// TIA Portal V19 export
FUNCTION_BLOCK "TYPIC_C103_BF_LSK"   // FB21, FBD
TITLE = TYPIC_C103_BF_LSK: Laagspanning koker
{ S7_Optimized_Access := 'TRUE' }
AUTHOR : OCOTECH
FAMILY : Typical
NAME : C103.801
// Logisch Object Besturing: C103.801
// 
// Het doel van de BF LSK (laagspanning koker) is om de algemene opvolging te voorzien van de laagspanningsinstallatie per verkeerskoker.
// stored: MemoryReserve 10, SetENOAutomatically false
   VAR_INPUT
      STU_ALG_LCK_SIG { ExternalAccessible := 'False'; ExternalVisible := 'False'; ExternalWritable := 'False'} : USInt;   // Onderdruk alarmen
   END_VAR
   VAR_IN_OUT
      VAR_REL : Array[0..1] of Bool;   // Array met de standmeldingen van alle vermogenschakelaars
   END_VAR
   VAR
      SIG { ExternalWritable := 'False'} : Struct   // Signaleringen
         AA01 : Bool;   // Laagspanningsinstallatie niet observeerbaar
         AA02 : Bool;   // Laagspanningsinstallatie storing algemeen
         A001 : Bool;   // Laagspanningsinstallatie standmelding beveiliging uit
         AB01 : Bool;   // Laagspanningsinstallatie niet beschikbaar
         AB02 : Bool;   // Laagspanningsinstallatie beperkt beschikbaar
      END_STRUCT;
      VAR { ExternalWritable := 'False'} : Struct   // Variabelen
         BSC : USInt;   // Geeft de beschikbaarheid aan van het deelsysteem
         LSK_STS : USInt;   // De status van het deelsysteem
         VGV_SIG_VOP : Bool;   // TRUE = Signaleringen vrijgegeven voor verkeersoperator FALSE = Onderdrukt
      END_STRUCT;
   END_VAR
BEGIN

REGION Network 1: START
END_REGION

REGION Network 2: +++ Bepalen beschikbaarheidsstatus +++
   // Beschikbaarheidsstatus (beschikbaar / beperkt beschikbaar / niet beschikbaar) bepalen.
END_REGION

REGION Network 3 (SCL): Beschikbaarheidsstatus bepalen
   IF 
       //voorwaarden "Niet beschikbaar"
       TRUE
   THEN
       //Beschikbaarheidsstatus = Niet Beschikbaar
       #VAR.BSC:= "NietBeschikbaar";
   ELSIF
       //voorwaarden "Beperkt beschikbaar"
       TRUE
   THEN
       //Beschikbaarheidsstatus = Beperkt Beschikbaar
       #VAR.BSC:= "Beperkt";
   ELSE
       //Beschikbaarheidsstatus = Beschikbaar
       #VAR.BSC:= "Beschikbaar";
   END_IF;
END_REGION

REGION Network 4: +++ Signaleringen +++
   // Aanmaken signaleringen
END_REGION

REGION Network 5: Signalering AB01 : Niet Beschikbaar
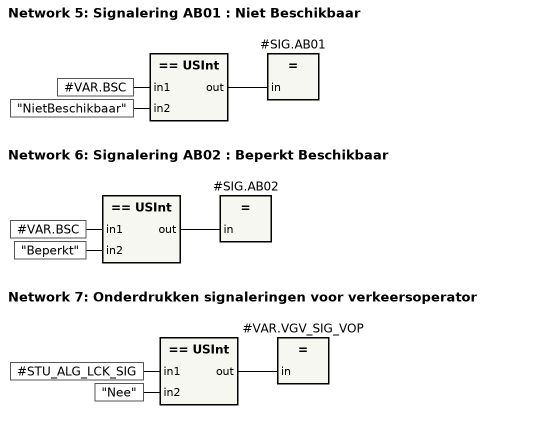
   #SIG.AB01 := #VAR.BSC = "NietBeschikbaar";
END_REGION

REGION Network 6: Signalering AB02 : Beperkt Beschikbaar
   #SIG.AB02 := #VAR.BSC = "Beperkt";
END_REGION

REGION Network 7: Onderdrukken signaleringen voor verkeersoperator
   // Via de variabele VGV_SIG_VOP wordt aan IRIS SCADA doorgegeven of signaleringen (bestemd voor de verkeersoperator) van de deze functie zichtbaar (of onderdrukt) moeten zijn.
   #VAR.VGV_SIG_VOP := #STU_ALG_LCK_SIG = "Nee";
END_REGION

REGION Network 8: +++ Doorkoppeling energieverbruik en vermogen LSK +++
   // De actuele vermogen en energiemeting wordt doorgegeven aan de coordinerende functie Energievoorziening.
END_REGION

REGION Network 9: EINDE
   // Variabelen van intern scada rakvlak naar outputs copieren
END_REGION
END_FUNCTION_BLOCK
